// Contains all the available path seperators based on the operating system.
{attribute 'no_explicit_call' := 'Body contains no logic, calling methods only allowed.'}
PROGRAM PathSeperator
VAR
END_VAR

// Returns system independent path separator "/"
PROPERTY SystemIndependent : ZigaLibs_Core.T_Char
GET
SystemIndependent := Windows;
END_GET
END_PROPERTY

// Returns UNIX path separator "\"
PROPERTY Unix : ZigaLibs_Core.T_Char
GET
Unix := '\';
END_GET
END_PROPERTY

// Returns WINDOWS path separator "/"
PROPERTY Windows : ZigaLibs_Core.T_Char
GET
Windows := '/';
END_GET
END_PROPERTY

END_PROGRAM

(* stored: Version 1.1.0.1, ProductVersion 3.1.4024.14
   POU PathSeperator: Id {ff96902c-5136-0ae0-1075-e89641639929}, SpecialFunc None
   Property SystemIndependent: Id {399b46e0-d2cc-0c27-2cf2-5a616d06b4ae}
   Get Get: Id {59fb9107-e1d6-083c-0654-ab20acbc5a56}
   Property Unix: Id {e97c3d91-3eab-0406-1364-8c28b8596b23}
   Get Get: Id {23e88559-d182-0fe2-2b74-4b158b9d61f7}
   Property Windows: Id {79e1fca6-79e7-07e8-052c-4d9c7cd66fd4}
   Get Get: Id {e5c4fede-1050-0288-3d07-af087dead439} *)
